{attribute 'qualified_only'}
{attribute 'strict'}
{attribute 'to_string'}
TYPE E_StsActState :
(
	StartupCheck,
	AssemblyCheck,
	Idle,
	DataLogging,
	RobotSlotHold,
	AngleAdj,
	PositionAdj,
	ProductMounting,
	ProductDisMounting,
	Disabled,
	Error,
	HoldForValveRelease
);
END_TYPE

(* stored: Version 1.1.0.1
   DUT E_StsActState: Id {265bdca5-8442-4554-9653-da45c5676766} *)
